// TIA Portal V18 export
FUNCTION_BLOCK "FS_VerticalBeam"   // FB5, F_LAD
{ S7_Optimized_Access := 'TRUE' }
VERSION : 0.1
// stored: AutoNumber false, IsIECCheckEnabled false, UDAEnableTagReadback false
   VAR_INPUT
      ACK : Bool;
   END_VAR
   VAR_OUTPUT
      ES_OK : Bool;
   END_VAR
   VAR
      EStop1 { S7_SetPoint := 'True'} : ESTOP1;
      EStop2 { S7_SetPoint := 'True'} : ESTOP1;
      EStop3 { S7_SetPoint := 'True'} : ESTOP1;
      EStop4 { S7_SetPoint := 'True'} : ESTOP1;
      door1 : SFDOOR;
      door2 : SFDOOR;
      Key : SFDOOR;
      KeyControl : SFDOOR;
   END_VAR
BEGIN

REGION Network 1: E-Stop1
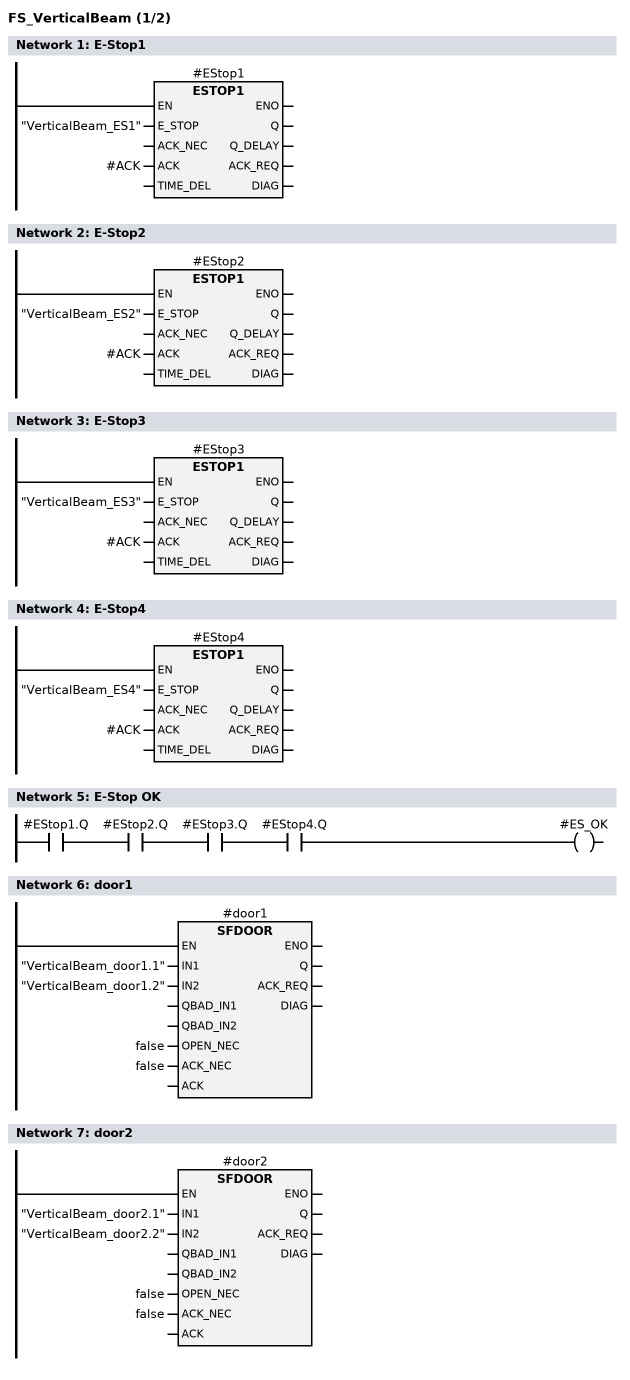
   RUNG wire#powerrail
      #EStop1.ESTOP1(E_STOP := "VerticalBeam_ES1", ACK_NEC :=, ACK := #ACK, TIME_DEL :=, Q =>, Q_DELAY =>, ACK_REQ =>, DIAG =>)
   END_RUNG
   // the same network as SCL:
   #EStop1(E_STOP := "VerticalBeam_ES1", ACK := #ACK);   // ESTOP1
END_REGION

REGION Network 2: E-Stop2
   RUNG wire#powerrail
      #EStop2.ESTOP1(E_STOP := "VerticalBeam_ES2", ACK_NEC :=, ACK := #ACK, TIME_DEL :=, Q =>, Q_DELAY =>, ACK_REQ =>, DIAG =>)
   END_RUNG
   // the same network as SCL:
   #EStop2(E_STOP := "VerticalBeam_ES2", ACK := #ACK);   // ESTOP1
END_REGION

REGION Network 3: E-Stop3
   RUNG wire#powerrail
      #EStop3.ESTOP1(E_STOP := "VerticalBeam_ES3", ACK_NEC :=, ACK := #ACK, TIME_DEL :=, Q =>, Q_DELAY =>, ACK_REQ =>, DIAG =>)
   END_RUNG
   // the same network as SCL:
   #EStop3(E_STOP := "VerticalBeam_ES3", ACK := #ACK);   // ESTOP1
END_REGION

REGION Network 4: E-Stop4
   RUNG wire#powerrail
      #EStop4.ESTOP1(E_STOP := "VerticalBeam_ES4", ACK_NEC :=, ACK := #ACK, TIME_DEL :=, Q =>, Q_DELAY =>, ACK_REQ =>, DIAG =>)
   END_RUNG
   // the same network as SCL:
   #EStop4(E_STOP := "VerticalBeam_ES4", ACK := #ACK);   // ESTOP1
END_REGION

REGION Network 5: E-Stop OK
   RUNG wire#powerrail
      Contact( #EStop1.Q )
      Contact( #EStop2.Q )
      Contact( #EStop3.Q )
      Contact( #EStop4.Q )
      Coil( #ES_OK )
   END_RUNG
   // the same network as SCL:
   #ES_OK := #EStop1.Q AND #EStop2.Q AND #EStop3.Q AND #EStop4.Q;
END_REGION

REGION Network 6: door1
   RUNG wire#powerrail
      #door1.SFDOOR(IN1 := "VerticalBeam_door1.1", IN2 := "VerticalBeam_door1.2", QBAD_IN1 :=, QBAD_IN2 :=, OPEN_NEC := false, ACK_NEC := false, ACK :=, Q =>, ACK_REQ =>, DIAG =>)
   END_RUNG
   // the same network as SCL:
   #door1(IN1 := "VerticalBeam_door1.1", IN2 := "VerticalBeam_door1.2", OPEN_NEC := false, ACK_NEC := false);   // SFDOOR
END_REGION

REGION Network 7: door2
   RUNG wire#powerrail
      #door2.SFDOOR(IN1 := "VerticalBeam_door2.1", IN2 := "VerticalBeam_door2.2", QBAD_IN1 :=, QBAD_IN2 :=, OPEN_NEC := false, ACK_NEC := false, ACK :=, Q =>, ACK_REQ =>, DIAG =>)
   END_RUNG
   // the same network as SCL:
   #door2(IN1 := "VerticalBeam_door2.1", IN2 := "VerticalBeam_door2.2", OPEN_NEC := false, ACK_NEC := false);   // SFDOOR
END_REGION

REGION Network 8: Key
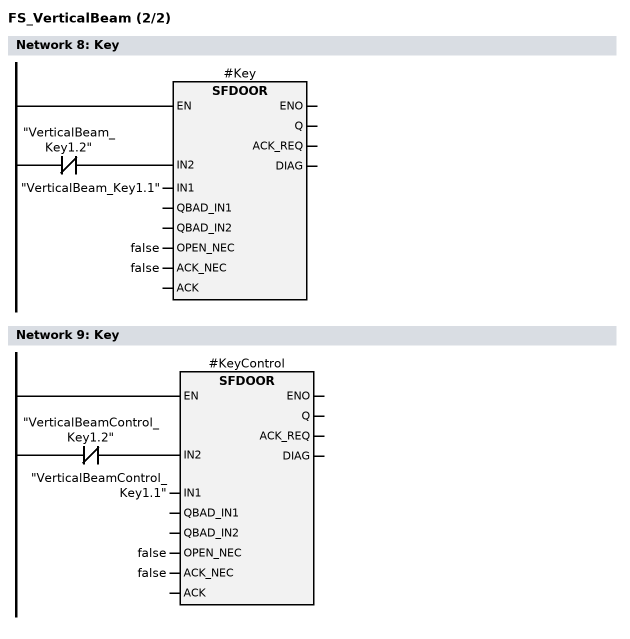
   RUNG wire#powerrail
      #Key.SFDOOR(IN2 := wire#w1, IN1 := "VerticalBeam_Key1.1", QBAD_IN1 :=, QBAD_IN2 :=, OPEN_NEC := false, ACK_NEC := false, ACK :=, Q =>, ACK_REQ =>, DIAG =>)
   END_RUNG
   RUNG wire#powerrail
      I_Contact( "VerticalBeam_Key1.2" )
   END_RUNG wire#w1
   // the same network as SCL:
   #Key(IN2 := NOT "VerticalBeam_Key1.2", IN1 := "VerticalBeam_Key1.1", OPEN_NEC := false, ACK_NEC := false);   // SFDOOR
END_REGION

REGION Network 9: Key
   RUNG wire#powerrail
      #KeyControl.SFDOOR(IN2 := wire#w1, IN1 := "VerticalBeamControl_Key1.1", QBAD_IN1 :=, QBAD_IN2 :=, OPEN_NEC := false, ACK_NEC := false, ACK :=, Q =>, ACK_REQ =>, DIAG =>)
   END_RUNG
   RUNG wire#powerrail
      I_Contact( "VerticalBeamControl_Key1.2" )
   END_RUNG wire#w1
   // the same network as SCL:
   #KeyControl(IN2 := NOT "VerticalBeamControl_Key1.2",   // SFDOOR
               IN1 := "VerticalBeamControl_Key1.1",
               OPEN_NEC := false,
               ACK_NEC := false);
END_REGION
END_FUNCTION_BLOCK
